FUNCTION FindYoungest : myPersonType
VAR_INPUT
	ListOfEmplyees:myEmployees;
END_VAR
VAR
	i: INT;
END_VAR

FindYoungest:=ListOfEmplyees[1];
FOR	i:=2	TO	SIZEOF(ListOfEmplyees)/SIZEOF(myPersonType)	DO
	IF	ListOfEmplyees[i].age>0	THEN
		IF	ListOfEmplyees[i].age<FindYoungest.age	THEN
			FindYoungest:=ListOfEmplyees[i];
		END_IF
	END_IF
END_FOR

END_FUNCTION

(* stored: Version 1.1.0.1, ProductVersion 3.1.4024.11
   POU FindYoungest: Id {0162a207-dc78-4efd-890e-9b28f4e5f3ea}, SpecialFunc None *)
